// TIA Portal V17 export
// export: Created 2021-12-03T08:12:53.1584196Z, ExportSetting WithDefaults, DisplayName Totally Integrated Automation Portal, DisplayVersion V17, DisplayName TIA Portal Openness, DisplayVersion V17, DisplayName TIA Portal Version Control Interface, DisplayVersion V17, DisplayName STEP 7 Professional, DisplayVersion V17, DisplayName STEP 7 Safety, DisplayVersion V17, DisplayName WinCC Advanced, DisplayVersion V17
DATA_BLOCK "GDB_HMI_IO_Retain"   // DB1004
VERSION : 0.1
// stored: AutoNumber false, IsOnlyStoredInLoadMemory false, IsWriteProtectedInAS false
   VAR RETAIN
      AccChiller : Struct   // Значения для чиллера ускорителя
         ChilPwrOnTm_PT : Int;   // Время подготовки чиллера мс
         ChilPwrOnTm_PT_ms : Time := T#0MS;   // Время подготовки чиллера мин
         ChilPwrOffTm_PT : Int;   // Время охлаждения чиллера мс
         ChilPwrOffTm_PT_ms : Time := T#0MS;   // Время охлаждения чиллера мин
         "Type" : Int;   // Тип ускорителя
      END_STRUCT;
      FrqConv : Struct
         FastSpeed : Int;
         LowSpeed : Int;
         Ramp : Int;
      END_STRUCT;
      "Version" : String := STRING#'Mini System V1.0';
      SensDist : Struct   // Расстояние между датчиками
         DistXRayFwdToXRayBwd : Int;   // Расстояние между датчиками XrayOnFwd и XrayOnBwd
      END_STRUCT;
      ScanSeqSet : Struct
         RfOn : Int;   // Время задержки в СВЧ
         RfOn_ms : Time;   // Время задержки в СВЧ мс
         XrayOn : Int;   // Время задержки в торм. излучении
         XrayOn_ms : Time;   // Время задержки в торм. излучении мс
         CycleTime : Int;   // Время для цикла
         CycleTime_ms : Time;   // Время для цикла, мс
      END_STRUCT;
      TmrValue : DInt;
   END_VAR
BEGIN
END_DATA_BLOCK
